Staubli VAL3: recvTrajPt.pgx

public program recvTrajPt(sio& x_sSocket (dimensions=1), num& x_nConnFlag (dimensions=1), RosSimpleMsg& x_msg (dimensions=1), bool& x_bFlag (dimensions=1))
begin
  // Copyright (c) 2016, Ocado Technology - Robotics Research Team
  // Copyright (c) 2021, Institute for Factory Automation and Production Systems (FAPS)
  //
  // Licensed under the Apache License, Version 2.0 (the "License");
  // you may not use this file except in compliance with the License.
  // You may obtain a copy of the License at
  //
  //     http://www.apache.org/licenses/LICENSE-2.0
  //
  // Unless required by applicable law or agreed to in writing, software
  // distributed under the License is distributed on an "AS IS" BASIS,
  // WITHOUT WARRANTIES OR CONDITIONS OF ANY KIND, either express or implied.
  // See the License for the specific language governing permissions and
  // limitations under the License.



  // attempt to receive message ID 11 data (prefix and header are in x_msg)
  rosTrajPtMsg.prefix.nLength=x_msg.prefix.nLength
  rosTrajPtMsg.header.nMsgType=x_msg.header.nMsgType
  rosTrajPtMsg.header.nCommType=x_msg.header.nCommType
  rosTrajPtMsg.header.nReplyCode=x_msg.header.nReplyCode

  call recvData(x_sSocket,rosTrajPtMsg.body.nData,x_nConnFlag,x_bFlag)
end
